Fanuc KAREL source: kd00001.KL

-- PROVISIONAL review KL for V770-1; original PC SHA256 6da1f5af4dc7b30b48aef21a2b824c57ba3b88f54666032e03dde12ab6853867
-- Incomplete behavior may be omitted. Consult companion uncertainty JSON. Do not deploy.
PROGRAM KD00001
%NOLOCKGROUP
VAR
  I : INTEGER
  J : INTEGER
  B : BOOLEAN
  R : REAL
  S : STRING[80]
BEGIN
  -- UNRESOLVED_PC offsets 5-12; opcodes 9D,23
  -- UNRESOLVED_PC offsets 17-21; opcodes 7F
END KD00001
